FUNCTION_BLOCK AlignValues (* Basic Function Block Type *)
  (* Standard: 61499-2 *)
  (* Version 0.0, 2011-12-18, 4DIAC-IDE, 4DIAC-Consortium *)
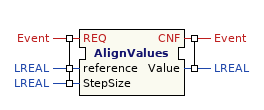
  EVENT_INPUT
    REQ WITH reference, StepSize;
  END_EVENT
  EVENT_OUTPUT
    CNF WITH Value; (* Execution Confirmation *)
  END_EVENT
  VAR_INPUT
    reference : LREAL;
    StepSize : LREAL;
  END_VAR
  VAR_OUTPUT
    Value : LREAL; (* Output event qualifier *)
  END_VAR
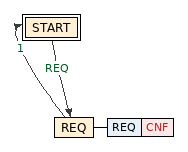
  EC_STATES
    START; (* Initial State *)
    REQ : REQ -> CNF; (* Normal execution *)
  END_STATES
  EC_TRANSITIONS
    START TO REQ := REQ;
    REQ TO START := 1;
  END_TRANSITIONS
  ALGORITHM REQ IN ST: (* Normally executed algorithm *)
	IF Value > reference + StepSize THEN

		Value := Value - StepSize;

	ELSIF Value < reference - StepSize THEN

		Value := Value + StepSize;

	ELSE

		Value := reference;


	END_IF
  END_ALGORITHM
END_FUNCTION_BLOCK
